// TwinCAT 3 PLC project Sample01
// ProgramVersion: 3.1.4020.10
// libraries:
//   Tc2_Standard, * (Beckhoff Automation GmbH)
//   Tc2_System, * (Beckhoff Automation GmbH)
//   Tc3_Module, * (Beckhoff Automation GmbH)
// project tree:
//   / PlcTask.TcTTO (not stored)
//   POUs/Commands/ FB_AirConComfortCommand.TcPOU (not stored), FB_AirConStandbyCommand.TcPOU (not stored), FB_LampSetLevelCommand.TcPOU (not stored), FB_MusicPlayCommand.TcPOU (not stored), FB_MusicStopCommand.TcPOU (not stored), FB_SocketOffCommand.TcPOU (not stored), FB_SocketOnCommand.TcPOU (not stored), I_Command.TcIO (not stored)
//   POUs/Invoker/ FB_SwitchPanel.TcPOU (not stored)
//   POUs/ MAIN.TcPOU (not stored)
//   POUs/Receiver/ FB_AirConditioning.TcPOU (not stored), FB_CDPlayer.TcPOU (not stored), FB_Lamp.TcPOU, FB_Socket.TcPOU (not stored)
// real-time tasks:
//   TASK PlcTask: cycle T#10ms, priority 20, ADS port 350

// ---- POUs/Receiver/FB_Lamp.TcPOU
FUNCTION_BLOCK PUBLIC FB_Lamp
VAR_OUTPUT
	byLevel			: BYTE;
END_VAR

PROPERTY PUBLIC Level : BYTE
GET
Level := byLevel;
END_GET
END_PROPERTY

METHOD PUBLIC SetLevel : BOOL
VAR_INPUT
	byNewLevel			: BYTE;
END_VAR
byLevel := byNewLevel;
END_METHOD

END_FUNCTION_BLOCK
